{attribute 'enable_dynamic_creation'}
FUNCTION_BLOCK FutureTimerBlink EXTENDS FB_AbstructFuture
VAR_INPUT
END_VAR
VAR_OUTPUT
END_VAR
VAR
	process_timer: TON;
	blink_timer: TON;
	_set_time :TIME;
	_result :UDINT;
	_output: REFERENCE TO BOOL;
	_process_time: TIME;
	_error_test :BOOL;
END_VAR

METHOD abort : BOOL
IF process_timer.IN THEN
	_set_time := process_timer.PT - process_timer.ET;
END_IF
process_timer(IN := FALSE);
_output := FALSE;
abort := TRUE;
END_METHOD

METHOD error_reset : BOOL // Must be overrided if future has any errors.
_error_test := FALSE;
_result := 0;
error_reset := TRUE;
END_METHOD

PROPERTY error_test : BOOL
SET
_error_test := error_test;
END_SET
END_PROPERTY

METHOD execute : BOOL
VAR_INPUT
END_VAR
blink_timer(IN := NOT blink_timer.Q, PT := T#0.5S);
IF _output AND blink_timer.Q THEN
	_output := FALSE;
ELSIF blink_timer.Q THEN
	_output := TRUE;
END_IF
process_timer(IN := TRUE,PT := _process_time);
execute := process_timer.Q;

IF _error_test THEN
	_result := 9;
	execute := TRUE;
END_IF
END_METHOD

METHOD init : BOOL
VAR_INPUT
END_VAR
_output := FALSE;
_set_time := _process_time;
process_timer(IN := FALSE);
blink_timer(IN := FALSE);
init := TRUE;
END_METHOD

PROPERTY nErrorID : HRESULT
GET
END_GET
END_PROPERTY

METHOD quit : BOOL
THIS^.init();
quit := TRUE;
END_METHOD

METHOD set_options : BOOL
VAR_INPUT
	error_test: BOOL;
END_VAR
_error_test := error_test;
END_METHOD

METHOD set_parameter : BOOL
VAR_INPUT
	process_time: TIME;
	output		: REFERENCE TO BOOL;
END_VAR
_process_time := process_time;
_output REF= output;
END_METHOD

END_FUNCTION_BLOCK

(* stored: Version 1.1.0.1, ProductVersion 3.1.4026.13
   POU FutureTimerBlink: Id {1076d71a-3a65-40e8-9c4e-a3e9e6fe7b78}, SpecialFunc None
   Method abort: Id {d02a02ce-eb9e-43cb-a107-d4fa0fc34c85}
   Method error_reset: Id {815d8bd7-31f0-4c03-b2f4-4d31f789f9df}
   Property error_test: Id {d9b3cf67-16cb-49d7-8b46-3414806d9c30}
   Set Set: Id {5564eced-c26d-425e-a4dd-cec087f3b7c5}
   Method execute: Id {a437ddec-c1d7-448f-a879-d2b8cfc9472f}
   Method init: Id {67f09d3d-5c6c-4b82-bc02-bd0d47e41f54}
   Property nErrorID: Id {d940a05b-457a-4571-af02-9c908c0ddd5a}
   Get Get: Id {f38a3ee9-4b95-4da3-b87d-09c08cdf31f1}
   Method quit: Id {906e42c6-5cb2-4ee4-be39-84be0bedded2}
   Method set_options: Id {0a1e520d-d945-4d73-90d6-0bff08014023}
   Method set_parameter: Id {591902e6-3324-4e1f-b5ae-fd9dd8b19019} *)
